Staubli VAL3: modelParmIdent.pjx

Parameters version=s7.9.1 stackSize=5000 millimeterUnit=true
Program file=modelParmIdent.pgx
Program file=start.pgx
Program file=stop.pgx
Data file=modelParmIdent.dtx
Type name=ModelParameter path=Disk://RobotController_Libs/ModelParameter/ModelParameter.pjx
